// TIA Portal V17 export
// export: Created 2024-09-02T12:49:54.3626857Z, ExportSetting WithDefaults, DisplayName Totally Integrated Automation Portal, DisplayVersion V17, DisplayName TIA Portal Openness, DisplayVersion V17, DisplayName TIA Portal Version Control Interface, DisplayVersion V17, DisplayName STEP 7 Professional, DisplayVersion V17, DisplayName STEP 7 Safety, DisplayVersion V17, DisplayName WinCC Professional, DisplayVersion V17
DATA_BLOCK "DB_F_ANW"   // DB7000, F_DB
TITLE = Safety
{ S7_Optimized_Access := 'TRUE'; DB_Accessible_From_OPC_UA := 'FALSE' }
AUTHOR : OlegFuehrus
FAMILY : SAFETY
NAME : SAFETY
VERSION : 0.1
// stored: AutoNumber false, DBAccessibleFromOPCUA false
   VAR
      QBAD : Bool;   // Baugruppenfehler / Assembly faults
      ACK_REQ : Bool;   // Quittierung Baugruppe erforderlich / acknowlege
      Res02 : Bool;
      Res03 : Bool;
      Res04 : Bool;
      Res05 : Bool;
      Res06 : Bool;
      Res07 : Bool;
      Fault_ack : Bool;   // Stoerung quittieren gesamt / Acknowledge fault total
      Fault_ack_01 : Bool;   // Stoerung quittieren / Acknowledge fault
      Fault_ack_02 : Bool;   // Stoerung quittieren / Acknowledge fault
      Fault_ack_03 : Bool;   // Stoerung quittieren / Acknowledge fault
      Fault_ack_04 : Bool;   // Stoerung quittieren / Acknowledge fault
      Fault_ack_05 : Bool;   // Stoerung quittieren / Acknowledge fault
      Fault_ack_06 : Bool;   // Stoerung quittieren / Acknowledge fault
      Fault_ack_07 : Bool;   // Stoerung quittieren / Acknowledge fault
      Fault_ack_08 : Bool;   // Stoerung quittieren / Acknowledge fault
      Fault_ack_09 : Bool;   // Stoerung quittieren / Acknowledge fault
      Fault_ack_10 : Bool;   // Stoerung quittieren / Acknowledge fault
      Fault_ack_11 : Bool;   // Stoerung quittieren / Acknowledge fault
      Fault_ack_12 : Bool;   // Stoerung quittieren / Acknowledge fault
      Fault_ack_13 : Bool;   // Stoerung quittieren / Acknowledge fault
      Fault_ack_14 : Bool;   // Stoerung quittieren / Acknowledge fault
      Fault_ack_15 : Bool;   // Stoerung quittieren / Acknowledge fault
      FP_Fault_ack : Bool;   // HM Stoerung quittieren gesamt / HM Acknowledge fault total
      FP_Fault_ack_01 : Bool;   // HM Stoerung quittieren / HM Acknowledge fault
      FP_Fault_ack_02 : Bool;   // HM Stoerung quittieren / HM Acknowledge fault
      FP_Fault_ack_03 : Bool;   // HM Stoerung quittieren / HM Acknowledge fault
      FP_Fault_ack_04 : Bool;   // HM Stoerung quittieren / HM Acknowledge fault
      FP_Fault_ack_05 : Bool;   // HM Stoerung quittieren / HM Acknowledge fault
      FP_Fault_ack_06 : Bool;   // HM Stoerung quittieren / HM Acknowledge fault
      FP_Fault_ack_07 : Bool;   // HM Stoerung quittieren / HM Acknowledge fault
      FP_Fault_ack_08 : Bool;   // HM Stoerung quittieren / HM Acknowledge fault
      FP_Fault_ack_09 : Bool;   // HM Stoerung quittieren / HM Acknowledge fault
      FP_Fault_ack_10 : Bool;   // HM Stoerung quittieren / HM Acknowledge fault
      FP_Fault_ack_11 : Bool;   // HM Stoerung quittieren / HM Acknowledge fault
      FP_Fault_ack_12 : Bool;   // HM Stoerung quittieren / HM Acknowledge fault
      FP_Fault_ack_13 : Bool;   // HM Stoerung quittieren / HM Acknowledge fault
      FP_Fault_ack_14 : Bool;   // HM Stoerung quittieren / HM Acknowledge fault
      FP_Fault_ack_15 : Bool;   // HM Stoerung quittieren / HM Acknowledge fault
      E_Stop : Bool;   // Not-Halt i.O. Anlage gesamt / Emergency stop OK. Total investment
      E_Stop_01 : Bool;   // NOT-Halt / emergency stop
      E_Stop_02 : Bool;   // NOT-Halt / emergency stop
      E_Stop_03 : Bool;   // NOT-Halt / emergency stop
      E_Stop_04 : Bool;   // NOT-Halt / emergency stop
      E_Stop_05 : Bool;   // NOT-Halt / emergency stop
      E_Stop_06 : Bool;   // NOT-Halt / emergency stop
      E_Stop_07 : Bool;   // NOT-Halt / emergency stop
      E_Stop_08 : Bool;   // NOT-Halt / emergency stop
      E_Stop_09 : Bool;   // NOT-Halt / emergency stop
      E_Stop_Delay : Bool;   // Not-Halt ausschaltverzögert gesamt / Emergency-stop off-delayed total
      E_Stop_Delay_01 : Bool;   // Not-Halt ausschaltverzögert / Emergency-stop off-delayed
      E_Stop_Delay_02 : Bool;   // Not-Halt ausschaltverzögert / Emergency-stop off-delayed
      E_Stop_Delay_03 : Bool;   // Not-Halt ausschaltverzögert / Emergency-stop off-delayed
      E_Stop_Delay_04 : Bool;   // Not-Halt ausschaltverzögert / Emergency-stop off-delayed
      E_Stop_Delay_05 : Bool;   // Not-Halt ausschaltverzögert / Emergency-stop off-delayed
      E_Stop_Delay_06 : Bool;   // Not-Halt ausschaltverzögert / Emergency-stop off-delayed
      E_Stop_Delay_07 : Bool;   // Not-Halt ausschaltverzögert / Emergency-stop off-delayed
      E_Stop_Delay_08 : Bool;   // Not-Halt ausschaltverzögert / Emergency-stop off-delayed
      E_Stop_Delay_09 : Bool;   // Not-Halt ausschaltverzögert / Emergency-stop off-delayed
      E_Stop_Req : Bool;   // Not-Halt Anforderung quittieren gesamt / Acknowledge emergency-stop request total
      E_Stop_Req_01 : Bool;   // Not-Halt Anforderung quittieren / Acknowledge emergency-stop request
      E_Stop_Req_02 : Bool;   // Not-Halt Anforderung quittieren / Acknowledge emergency-stop request
      E_Stop_Req_03 : Bool;   // Not-Halt Anforderung quittieren / Acknowledge emergency-stop request
      E_Stop_Req_04 : Bool;   // Not-Halt Anforderung quittieren / Acknowledge emergency-stop request
      E_Stop_Req_05 : Bool;   // Not-Halt Anforderung quittieren / Acknowledge emergency-stop request
      E_Stop_Req_06 : Bool;   // Not-Halt Anforderung quittieren / Acknowledge emergency-stop request
      E_Stop_Req_07 : Bool;   // Not-Halt Anforderung quittieren / Acknowledge emergency-stop request
      E_Stop_Req_08 : Bool;   // Not-Halt Anforderung quittieren / Acknowledge emergency-stop request
      E_Stop_Req_09 : Bool;   // Not-Halt Anforderung quittieren / Acknowledge emergency-stop request
      LC : Bool;   // Lichtgitter i.O. Anlage gesamt / Light grid o. k. Total investment
      LC_01 : Bool;   // Lichtgitter / light curtain
      LC_02 : Bool;   // Lichtgitter / light curtain
      LC_03 : Bool;   // Lichtgitter / light curtain
      LC_04 : Bool;   // Lichtgitter / light curtain
      LC_05 : Bool;   // Lichtgitter / light curtain
      LC_06 : Bool;   // Lichtgitter / light curtain
      LC_Req : Bool;   // Lichtgitter Anforderung quittieren gesamt / Light curtain acknowledge request total
      LC_Req_01 : Bool;   // Lichtgitter Anforderung quittieren / Light curtain acknowledge request
      LC_Req_02 : Bool;   // Lichtgitter Anforderung quittieren / Light curtain acknowledge request
      LC_Req_03 : Bool;   // Lichtgitter Anforderung quittieren / Light curtain acknowledge request
      LC_Req_04 : Bool;   // Lichtgitter Anforderung quittieren / Light curtain acknowledge request
      LC_Req_05 : Bool;   // Lichtgitter Anforderung quittieren / Light curtain acknowledge request
      LC_Req_06 : Bool;   // Lichtgitter Anforderung quittieren / Light curtain acknowledge request
      LC_Fault : Bool;   // Lichtgitter Überwachungskanal fehler gesamt / Light curtain monitoring channel total error
      LC_Fault_01 : Bool;   // Lichtgitter Überwachungskanal fehler / Light curtain monitoring channel error
      LC_Fault_02 : Bool;   // Lichtgitter Überwachungskanal fehler / Light curtain monitoring channel error
      LC_Fault_03 : Bool;   // Lichtgitter Überwachungskanal fehler / Light curtain monitoring channel error
      LC_Fault_04 : Bool;   // Lichtgitter Überwachungskanal fehler / Light curtain monitoring channel error
      LC_Fault_05 : Bool;   // Lichtgitter Überwachungskanal fehler / Light curtain monitoring channel error
      LC_Fault_06 : Bool;   // Lichtgitter Überwachungskanal fehler / Light curtain monitoring channel error
      LC_MUT : Bool;   // Lichtgitter Muting i.O. Anlage gesamt / Light curtain muting total investment OK
      LC_MUT_01 : Bool;   // Lichtgitter Muting Einlauf / Light curtain muting inlet
      LC_MUT_02 : Bool;   // Lichtgitter Muting Auslauf / Light curtain muting outlet
      LC_MUT_03 : Bool;   // Lichtgitter Muting i.O. Anlage / light curtain muting facility OK
      LC_MUT_04 : Bool;   // Lichtgitter Muting i.O. Anlage / light curtain muting facility OK
      LC_MUT_05 : Bool;   // Lichtgitter Muting i.O. Anlage / light curtain muting facility OK
      LC_MUT_06 : Bool;   // Lichtgitter Muting i.O. Anlage / light curtain muting facility OK
      LC_MUT_Muting : Bool;   // Lichtgitter Muting aktiv / Light curtain muting active
      LC_MUT_Muting_01 : Bool;   // Lichtgitter Muting Einlauf aktiv / Light curtain muting infeed active
      LC_MUT_Muting_02 : Bool;   // Lichtgitter Muting Auslauf aktiv / Light grid muting outlet active
      LC_MUT_Muting_03 : Bool;   // Lichtgitter Muting aktiv / Light curtain muting active
      LC_MUT_Muting_04 : Bool;   // Lichtgitter Muting aktiv / Light curtain muting active
      LC_MUT_Muting_05 : Bool;   // Lichtgitter Muting aktiv / Light curtain muting active
      LC_MUT_Muting_06 : Bool;   // Lichtgitter Muting aktiv / Light curtain muting active
      LC_MUT_Req : Bool;   // Lichtgitter Muting Anforderung quittieren / Confirm the request to mute the light curtain
      LC_MUT_Req_01 : Bool;   // Lichtgitter Muting Anforderung / Light curtain muting requirement
      LC_MUT_Req_02 : Bool;   // Lichtgitter Muting Anforderung / Light curtain muting requirement
      LC_MUT_Req_03 : Bool;   // Lichtgitter Muting Anforderung / Light curtain muting requirement
      LC_MUT_Req_04 : Bool;   // Lichtgitter Muting Anforderung / Light curtain muting requirement
      LC_MUT_Req_05 : Bool;   // Lichtgitter Muting Anforderung / Light curtain muting requirement
      LC_MUT_Req_06 : Bool;   // Lichtgitter Muting Anforderung / Light curtain muting requirement
      LC_MUT_Fault : Bool;   // Lichtgitter Muting Überwachungskanal fehler / Light curtain muting monitoring channel error
      LC_MUT_Fault_01 : Bool;   // Lichtgitter Muting Überwachungskanal / Light curtain muting monitoring channel
      LC_MUT_Fault_02 : Bool;   // Lichtgitter Muting Überwachungskanal / Light curtain muting monitoring channel
      LC_MUT_Fault_03 : Bool;   // Lichtgitter Muting Überwachungskanal / Light curtain muting monitoring channel
      LC_MUT_Fault_04 : Bool;   // Lichtgitter Muting Überwachungskanal / Light curtain muting monitoring channel
      LC_MUT_Fault_05 : Bool;   // Lichtgitter Muting Überwachungskanal / Light curtain muting monitoring channel
      LC_MUT_Fault_06 : Bool;   // Lichtgitter Muting Überwachungskanal / Light curtain muting monitoring channel
      SD : Bool;   // Schutzgitter i.O. Anlage gesamt / Safety Door OK
      SD_01 : Bool;   // Schutzgitter i.O. Anlage / Protective grille OK facility
      SD_02 : Bool;   // Schutzgitter i.O. Anlage / Protective grille OK facility
      SD_03 : Bool;   // Schutzgitter i.O. Anlage / Protective grille OK facility
      SD_04 : Bool;   // Schutzgitter i.O. Anlage / Protective grille OK facility
      SD_05 : Bool;   // Schutzgitter i.O. Anlage / Protective grille OK facility
      SD_06 : Bool;   // Schutzgitter i.O. Anlage / Protective grille OK facility
      SD_Req : Bool;   // Schutzgitter Anforderung quittieren gesamt / Protective grille Acknowledge request total
      SD_Req_01 : Bool;   // Schutzgitter Anforderung quittieren / Protective grille Acknowledge request
      SD_Req_02 : Bool;   // Schutzgitter Anforderung quittieren / Protective grille Acknowledge request
      SD_Req_03 : Bool;   // Schutzgitter Anforderung quittieren / Protective grille Acknowledge request
      SD_Req_04 : Bool;   // Schutzgitter Anforderung quittieren / Protective grille Acknowledge request
      SD_Req_05 : Bool;   // Schutzgitter Anforderung quittieren / Protective grille Acknowledge request
      SD_Req_06 : Bool;   // Schutzgitter Anforderung quittieren / Protective grille Acknowledge request
      BR : Bool;   // Überbrückung i.O. Anlage gesamt / Bridging OK Total investment
      BR_01 : Bool;   // Überbrückung i.O. Anlage / Bridging OK facility
      BR_02 : Bool;   // Überbrückung i.O. Anlage / Bridging OK facility
      BR_03 : Bool;   // Überbrückung i.O. Anlage / Bridging OK facility
      BR_04 : Bool;   // Überbrückung i.O. Anlage / Bridging OK facility
      BR_05 : Bool;   // Überbrückung i.O. Anlage / Bridging OK facility
      BR_06 : Bool;   // Überbrückung i.O. Anlage / Bridging OK facility
      BR_Req : Bool;   // Überbrückung Anforderung quittieren / Bypass Acknowledge request
      BR_Req_01 : Bool;   // Überbrückung Anforderung quittieren / Bypass Acknowledge request
      BR_Req_02 : Bool;   // Überbrückung Anforderung quittieren / Bypass Acknowledge request
      BR_Req_03 : Bool;   // Überbrückung Anforderung quittieren / Bypass Acknowledge request
      BR_Req_04 : Bool;   // Überbrückung Anforderung quittieren / Bypass Acknowledge request
      BR_Req_05 : Bool;   // Überbrückung Anforderung quittieren / Bypass Acknowledge request
      BR_Req_06 : Bool;   // Überbrückung Anforderung quittieren / Bypass Acknowledge request
      BR_Fault : Bool;   // Überbrückung Überwachungskanal fehler / Bypass Monitoring channel error
      BR_Fault_01 : Bool;   // Überbrückung Überwachungskanal fehler / Bypass Monitoring channel error
      BR_Fault_02 : Bool;   // Überbrückung Überwachungskanal fehler / Bypass Monitoring channel error
      BR_Fault_03 : Bool;   // Überbrückung Überwachungskanal fehler / Bypass Monitoring channel error
      BR_Fault_04 : Bool;   // Überbrückung Überwachungskanal fehler / Bypass Monitoring channel error
      BR_Fault_05 : Bool;   // Überbrückung Überwachungskanal fehler / Bypass Monitoring channel error
      BR_Fault_06 : Bool;   // Überbrückung Überwachungskanal fehler / Bypass Monitoring channel error
      ENBL : Bool;   // Freigabe Anlage gesamt / Total plant Approve
      ENBL_01 : Bool;   // Freigabe Anlage / Plant Approve
      ENBL_02 : Bool;   // Freigabe Anlage / Plant Approve
      ENBL_03 : Bool;   // Freigabe Anlage / Plant Approve
      ENBL_04 : Bool;   // Freigabe Anlage / Plant Approve
      ENBL_05 : Bool;   // Freigabe Anlage / Plant Approve
      ENBL_06 : Bool;   // Freigabe Anlage / Plant Approve
      ENBL_07 : Bool;   // Freigabe Anlage / Plant Approve
      ENBL_08 : Bool;   // Freigabe Anlage / Plant Approve
      ENBL_09 : Bool;   // Freigabe Anlage / Plant Approve
      ENBL_10 : Bool;   // Freigabe Anlage / Plant Approve
      ENBL_11 : Bool;   // Freigabe Anlage / Plant Approve
      ENBL_12 : Bool;   // Freigabe Anlage / Plant Approve
      ENBL_13 : Bool;   // Freigabe Anlage / Plant Approve
      ENBL_14 : Bool;   // Freigabe Anlage / Plant Approve
      ENBL_15 : Bool;   // Freigabe Anlage / Plant Approve
      ENBL_Delay : Bool;   // Freigabe Anlage Verzögert gesamt / Enable system Delayed total
      ENBL_01_Delay : Bool;   // Freigabe Anlage Verzögert / Enable System Delayed
      ENBL_02_Delay : Bool;   // Freigabe Anlage Verzögert / Enable System Delayed
      ENBL_03_Delay : Bool;   // Freigabe Anlage Verzögert / Enable System Delayed
      ENBL_04_Delay : Bool;   // Freigabe Anlage Verzögert / Enable System Delayed
      ENBL_05_Delay : Bool;   // Freigabe Anlage Verzögert / Enable System Delayed
      ENBL_06_Delay : Bool;   // Freigabe Anlage Verzögert / Enable System Delayed
      ENBL_07_Delay : Bool;   // Freigabe Anlage Verzögert / Enable System Delayed
      ENBL_08_Delay : Bool;   // Freigabe Anlage Verzögert / Enable System Delayed
      ENBL_09_Delay : Bool;   // Freigabe Anlage Verzögert / Enable System Delayed
      ENBL_10_Delay : Bool;   // Freigabe Anlage Verzögert / Enable System Delayed
      ENBL_11_Delay : Bool;   // Freigabe Anlage Verzögert / Enable System Delayed
      ENBL_12_Delay : Bool;   // Freigabe Anlage Verzögert / Enable System Delayed
      ENBL_13_Delay : Bool;   // Freigabe Anlage Verzögert / Enable System Delayed
      ENBL_14_Delay : Bool;   // Freigabe Anlage Verzögert / Enable System Delayed
      ENBL_15_Delay : Bool;   // Freigabe Anlage Verzögert / Enable System Delayed
      ENBL_Error : Bool;   // Freigabe Rückführkreisüberwachung fehler gesamt / Enable feedback loop monitoring total error
      ENBL_Error_01 : Bool;   // Freigabe Rückführkreisüberwachung fehler / Enable feedback loop monitoring error
      ENBL_Error_02 : Bool;   // Freigabe Rückführkreisüberwachung fehler / Enable feedback loop monitoring error
      ENBL_Error_03 : Bool;   // Freigabe Rückführkreisüberwachung fehler / Enable feedback loop monitoring error
      ENBL_Error_04 : Bool;   // Freigabe Rückführkreisüberwachung fehler / Enable feedback loop monitoring error
      ENBL_Error_05 : Bool;   // Freigabe Rückführkreisüberwachung fehler / Enable feedback loop monitoring error
      ENBL_Error_06 : Bool;   // Freigabe Rückführkreisüberwachung fehler / Enable feedback loop monitoring error
      ENBL_Error_07 : Bool;   // Freigabe Rückführkreisüberwachung fehler / Enable feedback loop monitoring error
      ENBL_Error_08 : Bool;   // Freigabe Rückführkreisüberwachung fehler / Enable feedback loop monitoring error
      ENBL_Error_09 : Bool;   // Freigabe Rückführkreisüberwachung fehler / Enable feedback loop monitoring error
      ENBL_Error_10 : Bool;   // Freigabe Rückführkreisüberwachung fehler / Enable feedback loop monitoring error
      ENBL_Error_11 : Bool;   // Freigabe Rückführkreisüberwachung fehler / Enable feedback loop monitoring error
      ENBL_Error_12 : Bool;   // Freigabe Rückführkreisüberwachung fehler / Enable feedback loop monitoring error
      ENBL_Error_13 : Bool;   // Freigabe Rückführkreisüberwachung fehler / Enable feedback loop monitoring error
      ENBL_Error_14 : Bool;   // Freigabe Rückführkreisüberwachung fehler / Enable feedback loop monitoring error
      ENBL_Error_15 : Bool;   // Freigabe Rückführkreisüberwachung fehler / Enable feedback loop monitoring error
      ENBL_Req : Bool;   // Freigabe Rückführkreisüberwachung Anforderung quittieren / Enable feedback loop monitoring Acknowledge request
      ENBL_Req_01 : Bool;   // Freigabe Rückführkreisüberwachung Anforderung / Enable feedback loop monitoring Request
      ENBL_Req_02 : Bool;   // Freigabe Rückführkreisüberwachung Anforderung / Enable feedback loop monitoring Request
      ENBL_Req_03 : Bool;   // Freigabe Rückführkreisüberwachung Anforderung / Enable feedback loop monitoring Request
      ENBL_Req_04 : Bool;   // Freigabe Rückführkreisüberwachung Anforderung / Enable feedback loop monitoring Request
      ENBL_Req_05 : Bool;   // Freigabe Rückführkreisüberwachung Anforderung / Enable feedback loop monitoring Request
      ENBL_Req_06 : Bool;   // Freigabe Rückführkreisüberwachung Anforderung / Enable feedback loop monitoring Request
      ENBL_Req_07 : Bool;   // Freigabe Rückführkreisüberwachung Anforderung / Enable feedback loop monitoring Request
      ENBL_Req_08 : Bool;   // Freigabe Rückführkreisüberwachung Anforderung / Enable feedback loop monitoring Request
      ENBL_Req_09 : Bool;   // Freigabe Rückführkreisüberwachung Anforderung / Enable feedback loop monitoring Request
      ENBL_Req_10 : Bool;   // Freigabe Rückführkreisüberwachung Anforderung / Enable feedback loop monitoring Request
      ENBL_Req_11 : Bool;   // Freigabe Rückführkreisüberwachung Anforderung / Enable feedback loop monitoring Request
      ENBL_Req_12 : Bool;   // Freigabe Rückführkreisüberwachung Anforderung / Enable feedback loop monitoring Request
      ENBL_Req_13 : Bool;   // Freigabe Rückführkreisüberwachung Anforderung / Enable feedback loop monitoring Request
      ENBL_Req_14 : Bool;   // Freigabe Rückführkreisüberwachung Anforderung / Enable feedback loop monitoring Request
      ENBL_Req_15 : Bool;   // Freigabe Rückführkreisüberwachung Anforderung / Enable feedback loop monitoring Request
      SZ : Bool;   // Schutzbereich i.O. Anlage gesamt / Protection range OK facility total
      SZ_01 : Bool;   // Schutzbereich i.O. Anlage / Protection range OK facility
      SZ_02 : Bool;   // Schutzbereich i.O. Anlage / Protection range OK facility
      SZ_03 : Bool;   // Schutzbereich i.O. Anlage / Protection range OK facility
      SZ_04 : Bool;   // Schutzbereich i.O. Anlage / Protection range OK facility
      SZ_05 : Bool;   // Schutzbereich i.O. Anlage / Protection range OK facility
      SZ_06 : Bool;   // Schutzbereich i.O. Anlage / Protection range OK facility
      SZ_Req : Bool;   // Schtuzbereich Anforderung quittieren gesamt / Protection range Acknowledge request total
      SZ_Req_01 : Bool;   // Schtuzbereich Anforderung quittieren / Protection range Acknowledge request
      SZ_Req_02 : Bool;   // Schtuzbereich Anforderung quittieren / Protection range Acknowledge request
      SZ_Req_03 : Bool;   // Schtuzbereich Anforderung quittieren / Protection range Acknowledge request
      SZ_Req_04 : Bool;   // Schtuzbereich Anforderung quittieren / Protection range Acknowledge request
      SZ_Req_05 : Bool;   // Schtuzbereich Anforderung quittieren / Protection range Acknowledge request
      SZ_Req_06 : Bool;   // Schtuzbereich Anforderung quittieren / Protection range Acknowledge request
      SZ_Fault : Bool;   // Schutzbereich Überwachungskanal fehler gesamt / Protection zone Monitoring channel error total
      SZ_Fault_01 : Bool;   // Schutzbereich Überwachungskanal fehler / Protection zone Monitoring channel error
      SZ_Fault_02 : Bool;   // Schutzbereich Überwachungskanal fehler / Protection zone Monitoring channel error
      SZ_Fault_03 : Bool;   // Schutzbereich Überwachungskanal fehler / Protection zone Monitoring channel error
      SZ_Fault_04 : Bool;   // Schutzbereich Überwachungskanal fehler / Protection zone Monitoring channel error
      SZ_Fault_05 : Bool;   // Schutzbereich Überwachungskanal fehler / Protection zone Monitoring channel error
      SZ_Fault_06 : Bool;   // Schutzbereich Überwachungskanal fehler / Protection zone Monitoring channel error
      ENBL_Active : Bool;   // Freigabe Anlage gesamt / Total plant Approve
      ENBL_Active_01 : Bool;   // Freigabe / Approve
      ENBL_Active_02 : Bool;   // Freigabe / Approve
      ENBL_Active_03 : Bool;   // Freigabe / Approve
      ENBL_Active_04 : Bool;   // Freigabe / Approve
      ENBL_Active_05 : Bool;   // Freigabe / Approve
      ENBL_Active_06 : Bool;   // Freigabe / Approve
      ENBL_Active_07 : Bool;   // Freigabe / Approve
      ENBL_Active_08 : Bool;   // Freigabe / Approve
      ENBL_Active_09 : Bool;   // Freigabe / Approve
      ENBL_Active_10 : Bool;   // Freigabe / Approve
      ENBL_Active_11 : Bool;   // Freigabe / Approve
      ENBL_Active_12 : Bool;   // Freigabe / Approve
      ENBL_Active_13 : Bool;   // Freigabe / Approve
      ENBL_Active_14 : Bool;   // Freigabe / Approve
      ENBL_Active_15 : Bool;   // Freigabe / Approve
      ENBL_Rob_SD { ExternalWritable := 'False'} : Bool;   // Freigabe Schutztuer (nur eine offen) / Enable safety door (only one open)
      ENBL_Rob_E2 { ExternalWritable := 'False'} : Bool;   // Freigabe E2 (nur eine aktiv) / Enable E2 (only one active)
   END_VAR
BEGIN
END_DATA_BLOCK
